// TIA Portal V19 export
FUNCTION "AI SCALING" : Void   // FC5, LAD
{ S7_Optimized_Access := 'TRUE' }
// stored: SetENOAutomatically false
   VAR_TEMP   // added for the SCL form of the ladder/FBD networks
      _w1 : Bool;
   END_VAR
BEGIN

REGION Network 1: LEVEL TRANSMITTER-101 ANALOG
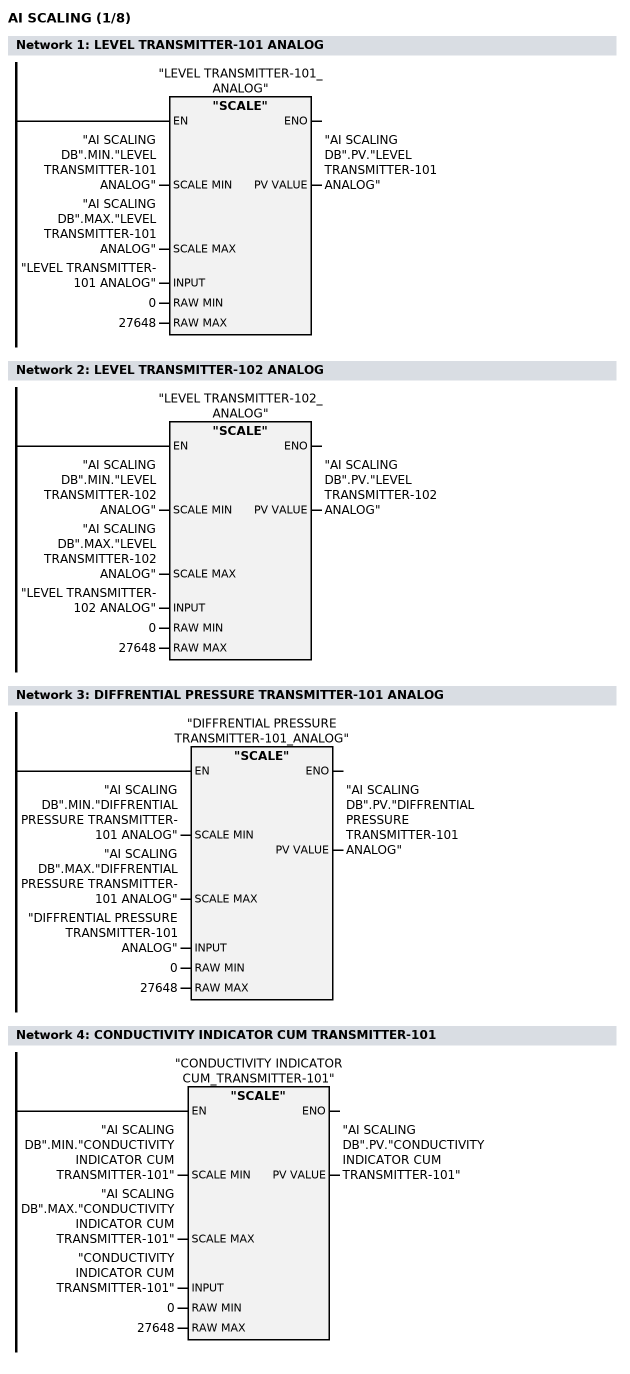
   RUNG wire#powerrail
      "LEVEL TRANSMITTER-101_ANALOG"("SCALE MIN" := "AI SCALING DB".MIN."LEVEL TRANSMITTER-101 ANALOG", "SCALE MAX" := "AI SCALING DB".MAX."LEVEL TRANSMITTER-101 ANALOG", INPUT := "LEVEL TRANSMITTER-101 ANALOG", "RAW MIN" := 0, "RAW MAX" := 27648, "PV VALUE" => "AI SCALING DB".PV."LEVEL TRANSMITTER-101 ANALOG")
   END_RUNG
   // the same network as SCL:
   "LEVEL TRANSMITTER-101_ANALOG"("SCALE MIN" := "AI SCALING DB".MIN."LEVEL TRANSMITTER-101 ANALOG",   // "SCALE"
                           "SCALE MAX" := "AI SCALING DB".MAX."LEVEL TRANSMITTER-101 ANALOG",
                           INPUT := "LEVEL TRANSMITTER-101 ANALOG",
                           "RAW MIN" := 0,
                           "RAW MAX" := 27648,
                           "PV VALUE" => "AI SCALING DB".PV."LEVEL TRANSMITTER-101 ANALOG");
END_REGION

REGION Network 2: LEVEL TRANSMITTER-102 ANALOG
   RUNG wire#powerrail
      "LEVEL TRANSMITTER-102_ANALOG"("SCALE MIN" := "AI SCALING DB".MIN."LEVEL TRANSMITTER-102 ANALOG", "SCALE MAX" := "AI SCALING DB".MAX."LEVEL TRANSMITTER-102 ANALOG", INPUT := "LEVEL TRANSMITTER-102 ANALOG", "RAW MIN" := 0, "RAW MAX" := 27648, "PV VALUE" => "AI SCALING DB".PV."LEVEL TRANSMITTER-102 ANALOG")
   END_RUNG
   // the same network as SCL:
   "LEVEL TRANSMITTER-102_ANALOG"("SCALE MIN" := "AI SCALING DB".MIN."LEVEL TRANSMITTER-102 ANALOG",   // "SCALE"
                           "SCALE MAX" := "AI SCALING DB".MAX."LEVEL TRANSMITTER-102 ANALOG",
                           INPUT := "LEVEL TRANSMITTER-102 ANALOG",
                           "RAW MIN" := 0,
                           "RAW MAX" := 27648,
                           "PV VALUE" => "AI SCALING DB".PV."LEVEL TRANSMITTER-102 ANALOG");
END_REGION

REGION Network 3: DIFFRENTIAL PRESSURE TRANSMITTER-101 ANALOG
   RUNG wire#powerrail
      "DIFFRENTIAL PRESSURE TRANSMITTER-101_ANALOG"("SCALE MIN" := "AI SCALING DB".MIN."DIFFRENTIAL PRESSURE TRANSMITTER-101 ANALOG", "SCALE MAX" := "AI SCALING DB".MAX."DIFFRENTIAL PRESSURE TRANSMITTER-101 ANALOG", INPUT := "DIFFRENTIAL PRESSURE TRANSMITTER-101 ANALOG", "RAW MIN" := 0, "RAW MAX" := 27648, "PV VALUE" => "AI SCALING DB".PV."DIFFRENTIAL PRESSURE TRANSMITTER-101 ANALOG")
   END_RUNG
   // the same network as SCL:
   "DIFFRENTIAL PRESSURE TRANSMITTER-101_ANALOG"("SCALE MIN" := "AI SCALING DB".MIN."DIFFRENTIAL PRESSURE TRANSMITTER-101 ANALOG",   // "SCALE"
                           "SCALE MAX" := "AI SCALING DB".MAX."DIFFRENTIAL PRESSURE TRANSMITTER-101 ANALOG",
                           INPUT := "DIFFRENTIAL PRESSURE TRANSMITTER-101 ANALOG",
                           "RAW MIN" := 0,
                           "RAW MAX" := 27648,
                           "PV VALUE" => "AI SCALING DB".PV."DIFFRENTIAL PRESSURE TRANSMITTER-101 ANALOG");
END_REGION

REGION Network 4: CONDUCTIVITY INDICATOR CUM TRANSMITTER-101
   RUNG wire#powerrail
      "CONDUCTIVITY INDICATOR CUM_TRANSMITTER-101"("SCALE MIN" := "AI SCALING DB".MIN."CONDUCTIVITY INDICATOR CUM TRANSMITTER-101", "SCALE MAX" := "AI SCALING DB".MAX."CONDUCTIVITY INDICATOR CUM TRANSMITTER-101", INPUT := "CONDUCTIVITY INDICATOR CUM TRANSMITTER-101", "RAW MIN" := 0, "RAW MAX" := 27648, "PV VALUE" => "AI SCALING DB".PV."CONDUCTIVITY INDICATOR CUM TRANSMITTER-101")
   END_RUNG
   // the same network as SCL:
   "CONDUCTIVITY INDICATOR CUM_TRANSMITTER-101"("SCALE MIN" := "AI SCALING DB".MIN."CONDUCTIVITY INDICATOR CUM TRANSMITTER-101",   // "SCALE"
                           "SCALE MAX" := "AI SCALING DB".MAX."CONDUCTIVITY INDICATOR CUM TRANSMITTER-101",
                           INPUT := "CONDUCTIVITY INDICATOR CUM TRANSMITTER-101",
                           "RAW MIN" := 0,
                           "RAW MAX" := 27648,
                           "PV VALUE" => "AI SCALING DB".PV."CONDUCTIVITY INDICATOR CUM TRANSMITTER-101");
END_REGION

REGION Network 5: DIFFRENTIAL PRESSURE TRANSMITTER-201
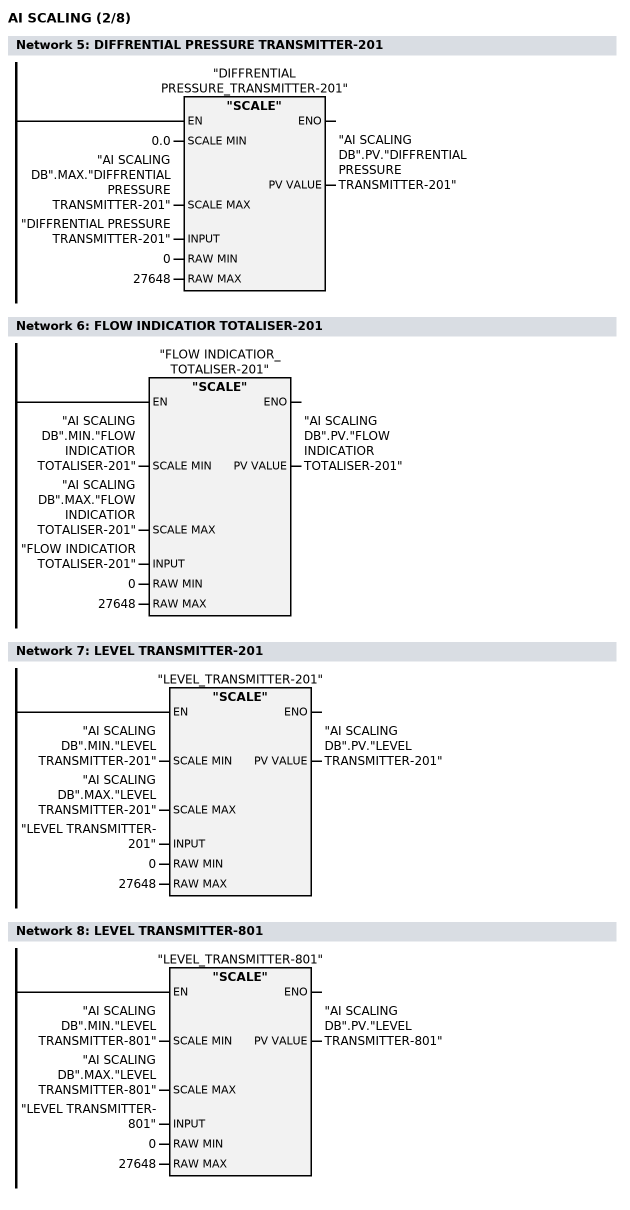
   RUNG wire#powerrail
      "DIFFRENTIAL PRESSURE_TRANSMITTER-201"("SCALE MIN" := 0.0, "SCALE MAX" := "AI SCALING DB".MAX."DIFFRENTIAL PRESSURE TRANSMITTER-201", INPUT := "DIFFRENTIAL PRESSURE TRANSMITTER-201", "RAW MIN" := 0, "RAW MAX" := 27648, "PV VALUE" => "AI SCALING DB".PV."DIFFRENTIAL PRESSURE TRANSMITTER-201")
   END_RUNG
   // the same network as SCL:
   "DIFFRENTIAL PRESSURE_TRANSMITTER-201"("SCALE MIN" := 0.0,   // "SCALE"
                           "SCALE MAX" := "AI SCALING DB".MAX."DIFFRENTIAL PRESSURE TRANSMITTER-201",
                           INPUT := "DIFFRENTIAL PRESSURE TRANSMITTER-201",
                           "RAW MIN" := 0,
                           "RAW MAX" := 27648,
                           "PV VALUE" => "AI SCALING DB".PV."DIFFRENTIAL PRESSURE TRANSMITTER-201");
END_REGION

REGION Network 6: FLOW INDICATIOR TOTALISER-201
   RUNG wire#powerrail
      "FLOW INDICATIOR_TOTALISER-201"("SCALE MIN" := "AI SCALING DB".MIN."FLOW INDICATIOR TOTALISER-201", "SCALE MAX" := "AI SCALING DB".MAX."FLOW INDICATIOR TOTALISER-201", INPUT := "FLOW INDICATIOR TOTALISER-201", "RAW MIN" := 0, "RAW MAX" := 27648, "PV VALUE" => "AI SCALING DB".PV."FLOW INDICATIOR TOTALISER-201")
   END_RUNG
   // the same network as SCL:
   "FLOW INDICATIOR_TOTALISER-201"("SCALE MIN" := "AI SCALING DB".MIN."FLOW INDICATIOR TOTALISER-201",   // "SCALE"
                           "SCALE MAX" := "AI SCALING DB".MAX."FLOW INDICATIOR TOTALISER-201",
                           INPUT := "FLOW INDICATIOR TOTALISER-201",
                           "RAW MIN" := 0,
                           "RAW MAX" := 27648,
                           "PV VALUE" => "AI SCALING DB".PV."FLOW INDICATIOR TOTALISER-201");
END_REGION

REGION Network 7: LEVEL TRANSMITTER-201
   RUNG wire#powerrail
      "LEVEL_TRANSMITTER-201"("SCALE MIN" := "AI SCALING DB".MIN."LEVEL TRANSMITTER-201", "SCALE MAX" := "AI SCALING DB".MAX."LEVEL TRANSMITTER-201", INPUT := "LEVEL TRANSMITTER-201", "RAW MIN" := 0, "RAW MAX" := 27648, "PV VALUE" => "AI SCALING DB".PV."LEVEL TRANSMITTER-201")
   END_RUNG
   // the same network as SCL:
   "LEVEL_TRANSMITTER-201"("SCALE MIN" := "AI SCALING DB".MIN."LEVEL TRANSMITTER-201",   // "SCALE"
                           "SCALE MAX" := "AI SCALING DB".MAX."LEVEL TRANSMITTER-201",
                           INPUT := "LEVEL TRANSMITTER-201",
                           "RAW MIN" := 0,
                           "RAW MAX" := 27648,
                           "PV VALUE" => "AI SCALING DB".PV."LEVEL TRANSMITTER-201");
END_REGION

REGION Network 8: LEVEL TRANSMITTER-801
   RUNG wire#powerrail
      "LEVEL_TRANSMITTER-801"("SCALE MIN" := "AI SCALING DB".MIN."LEVEL TRANSMITTER-801", "SCALE MAX" := "AI SCALING DB".MAX."LEVEL TRANSMITTER-801", INPUT := "LEVEL TRANSMITTER-801", "RAW MIN" := 0, "RAW MAX" := 27648, "PV VALUE" => "AI SCALING DB".PV."LEVEL TRANSMITTER-801")
   END_RUNG
   // the same network as SCL:
   "LEVEL_TRANSMITTER-801"("SCALE MIN" := "AI SCALING DB".MIN."LEVEL TRANSMITTER-801",   // "SCALE"
                           "SCALE MAX" := "AI SCALING DB".MAX."LEVEL TRANSMITTER-801",
                           INPUT := "LEVEL TRANSMITTER-801",
                           "RAW MIN" := 0,
                           "RAW MAX" := 27648,
                           "PV VALUE" => "AI SCALING DB".PV."LEVEL TRANSMITTER-801");
END_REGION

REGION Network 9: RESISTIVITY CUM TRANSMITTER 601
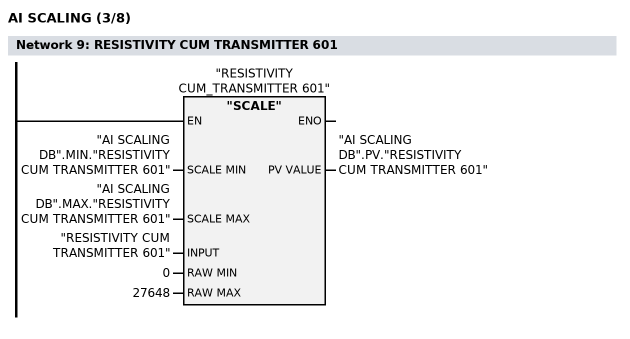
   RUNG wire#powerrail
      "RESISTIVITY CUM_TRANSMITTER 601"("SCALE MIN" := "AI SCALING DB".MIN."RESISTIVITY CUM TRANSMITTER 601", "SCALE MAX" := "AI SCALING DB".MAX."RESISTIVITY CUM TRANSMITTER 601", INPUT := "RESISTIVITY CUM TRANSMITTER 601", "RAW MIN" := 0, "RAW MAX" := 27648, "PV VALUE" => "AI SCALING DB".PV."RESISTIVITY CUM TRANSMITTER 601")
   END_RUNG
   // the same network as SCL:
   "RESISTIVITY CUM_TRANSMITTER 601"("SCALE MIN" := "AI SCALING DB".MIN."RESISTIVITY CUM TRANSMITTER 601",   // "SCALE"
                           "SCALE MAX" := "AI SCALING DB".MAX."RESISTIVITY CUM TRANSMITTER 601",
                           INPUT := "RESISTIVITY CUM TRANSMITTER 601",
                           "RAW MIN" := 0,
                           "RAW MAX" := 27648,
                           "PV VALUE" => "AI SCALING DB".PV."RESISTIVITY CUM TRANSMITTER 601");
END_REGION

REGION Network 10: PRESSURE TRANSMITTER 601
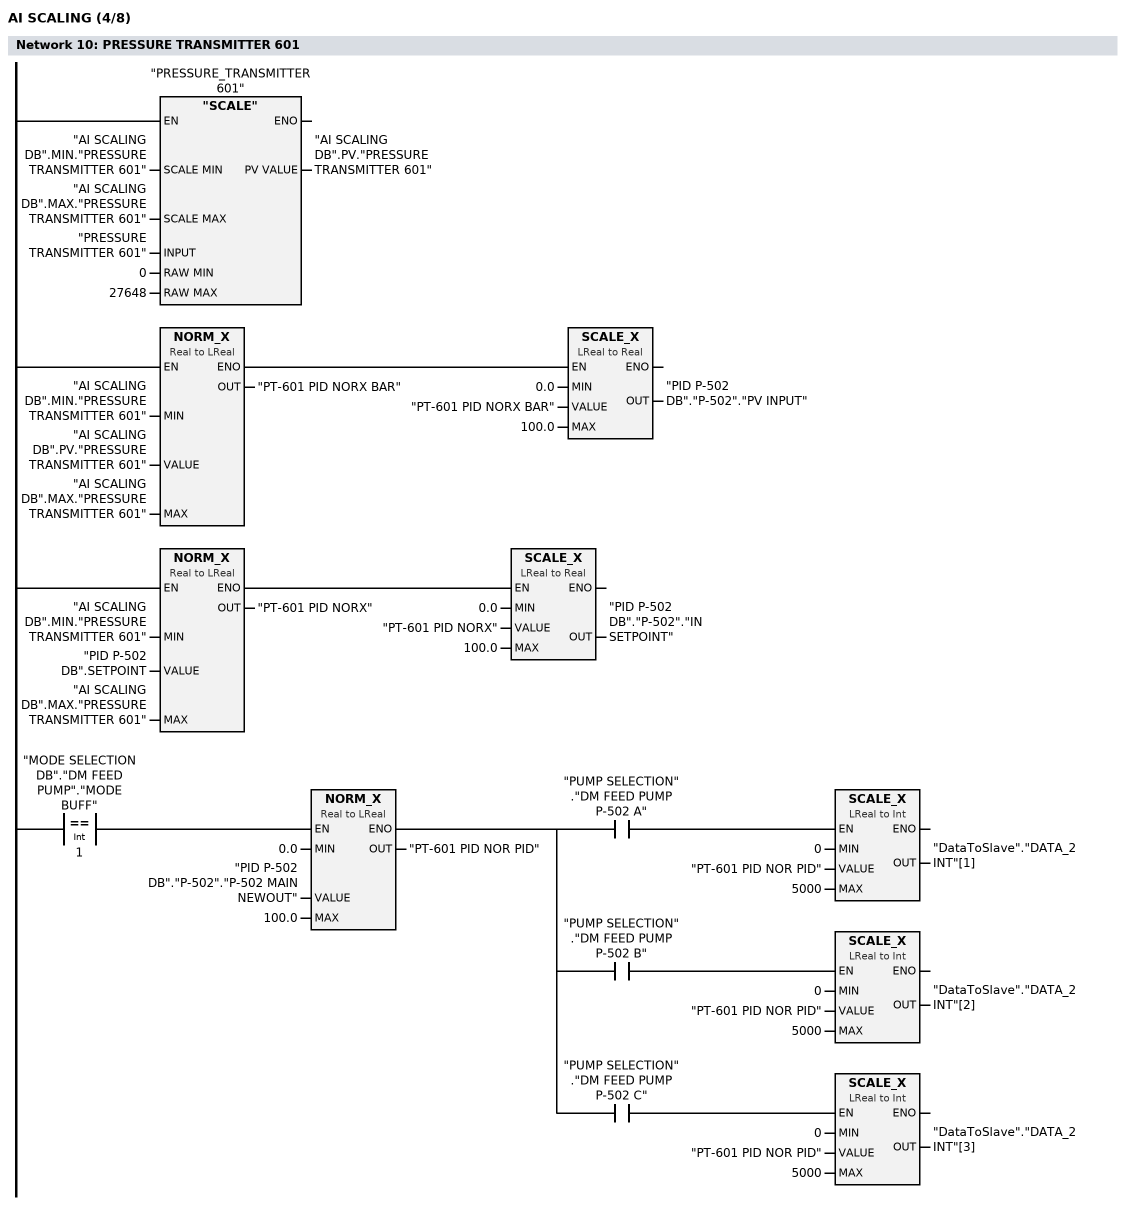
   RUNG wire#powerrail
      "PRESSURE_TRANSMITTER 601"("SCALE MIN" := "AI SCALING DB".MIN."PRESSURE TRANSMITTER 601", "SCALE MAX" := "AI SCALING DB".MAX."PRESSURE TRANSMITTER 601", INPUT := "PRESSURE TRANSMITTER 601", "RAW MIN" := 0, "RAW MAX" := 27648, "PV VALUE" => "AI SCALING DB".PV."PRESSURE TRANSMITTER 601")
   END_RUNG
   RUNG wire#powerrail
      { S7_Templates := "[SrcType := Real, DestType := LReal]" } Normalize(min := "AI SCALING DB".MIN."PRESSURE TRANSMITTER 601", value := "AI SCALING DB".PV."PRESSURE TRANSMITTER 601", max := "AI SCALING DB".MAX."PRESSURE TRANSMITTER 601", out => "PT-601 PID NORX BAR")
      { S7_Templates := "[SrcType := LReal, DestType := Real]" } Scale(min := 0.0, value := "PT-601 PID NORX BAR", max := 100.0, out => "PID P-502 DB"."P-502"."PV INPUT")
   END_RUNG
   RUNG wire#powerrail
      { S7_Templates := "[SrcType := Real, DestType := LReal]" } Normalize(min := "AI SCALING DB".MIN."PRESSURE TRANSMITTER 601", value := "PID P-502 DB".SETPOINT, max := "AI SCALING DB".MAX."PRESSURE TRANSMITTER 601", out => "PT-601 PID NORX")
      { S7_Templates := "[SrcType := LReal, DestType := Real]" } Scale(min := 0.0, value := "PT-601 PID NORX", max := 100.0, out => "PID P-502 DB"."P-502"."IN SETPOINT")
   END_RUNG
   RUNG wire#powerrail
      { S7_Templates := "SrcType := Int" } EQ_Contact(in1 := "MODE SELECTION DB"."DM FEED PUMP"."MODE BUFF", in2 := 1)
      { S7_Templates := "[SrcType := Real, DestType := LReal]" } Normalize(min := 0.0, value := "PID P-502 DB"."P-502"."P-502 MAIN NEWOUT", max := 100.0, out => "PT-601 PID NOR PID")
      wire#w1
      Contact( "PUMP SELECTION"."DM FEED PUMP P-502 A" )
      { S7_Templates := "[SrcType := LReal, DestType := Int]" } Scale(min := 0, value := "PT-601 PID NOR PID", max := 5000, out => "DataToSlave"."DATA_2 INT"[1])
   END_RUNG
   RUNG wire#w1
      Contact( "PUMP SELECTION"."DM FEED PUMP P-502 B" )
      { S7_Templates := "[SrcType := LReal, DestType := Int]" } Scale(min := 0, value := "PT-601 PID NOR PID", max := 5000, out => "DataToSlave"."DATA_2 INT"[2])
   END_RUNG
   RUNG wire#w1
      Contact( "PUMP SELECTION"."DM FEED PUMP P-502 C" )
      { S7_Templates := "[SrcType := LReal, DestType := Int]" } Scale(min := 0, value := "PT-601 PID NOR PID", max := 5000, out => "DataToSlave"."DATA_2 INT"[3])
   END_RUNG
   // the same network as SCL:
   "PRESSURE_TRANSMITTER 601"("SCALE MIN" := "AI SCALING DB".MIN."PRESSURE TRANSMITTER 601",   // "SCALE"
                           "SCALE MAX" := "AI SCALING DB".MAX."PRESSURE TRANSMITTER 601",
                           INPUT := "PRESSURE TRANSMITTER 601",
                           "RAW MIN" := 0,
                           "RAW MAX" := 27648,
                           "PV VALUE" => "AI SCALING DB".PV."PRESSURE TRANSMITTER 601");
   "PT-601 PID NORX BAR" := NORM_X(MIN := "AI SCALING DB".MIN."PRESSURE TRANSMITTER 601", VALUE := "AI SCALING DB".PV."PRESSURE TRANSMITTER 601", MAX := "AI SCALING DB".MAX."PRESSURE TRANSMITTER 601");
   "PID P-502 DB"."P-502"."PV INPUT" := SCALE_X(MIN := 0.0, VALUE := "PT-601 PID NORX BAR", MAX := 100.0);
   "PT-601 PID NORX" := NORM_X(MIN := "AI SCALING DB".MIN."PRESSURE TRANSMITTER 601", VALUE := "PID P-502 DB".SETPOINT, MAX := "AI SCALING DB".MAX."PRESSURE TRANSMITTER 601");
   "PID P-502 DB"."P-502"."IN SETPOINT" := SCALE_X(MIN := 0.0, VALUE := "PT-601 PID NORX", MAX := 100.0);
   #_w1 := "MODE SELECTION DB"."DM FEED PUMP"."MODE BUFF" = 1;
   IF #_w1 THEN
       "PT-601 PID NOR PID" := NORM_X(MIN := 0.0, VALUE := "PID P-502 DB"."P-502"."P-502 MAIN NEWOUT", MAX := 100.0);
   END_IF;
   IF #_w1 AND "PUMP SELECTION"."DM FEED PUMP P-502 A" THEN
       "DataToSlave"."DATA_2 INT"[1] := SCALE_X(MIN := 0, VALUE := "PT-601 PID NOR PID", MAX := 5000);
   END_IF;
   IF #_w1 AND "PUMP SELECTION"."DM FEED PUMP P-502 B" THEN
       "DataToSlave"."DATA_2 INT"[2] := SCALE_X(MIN := 0, VALUE := "PT-601 PID NOR PID", MAX := 5000);
   END_IF;
   IF #_w1 AND "PUMP SELECTION"."DM FEED PUMP P-502 C" THEN
       "DataToSlave"."DATA_2 INT"[3] := SCALE_X(MIN := 0, VALUE := "PT-601 PID NOR PID", MAX := 5000);
   END_IF;
END_REGION

REGION Network 11: FLOW INDICATIOR TOTALISER 601
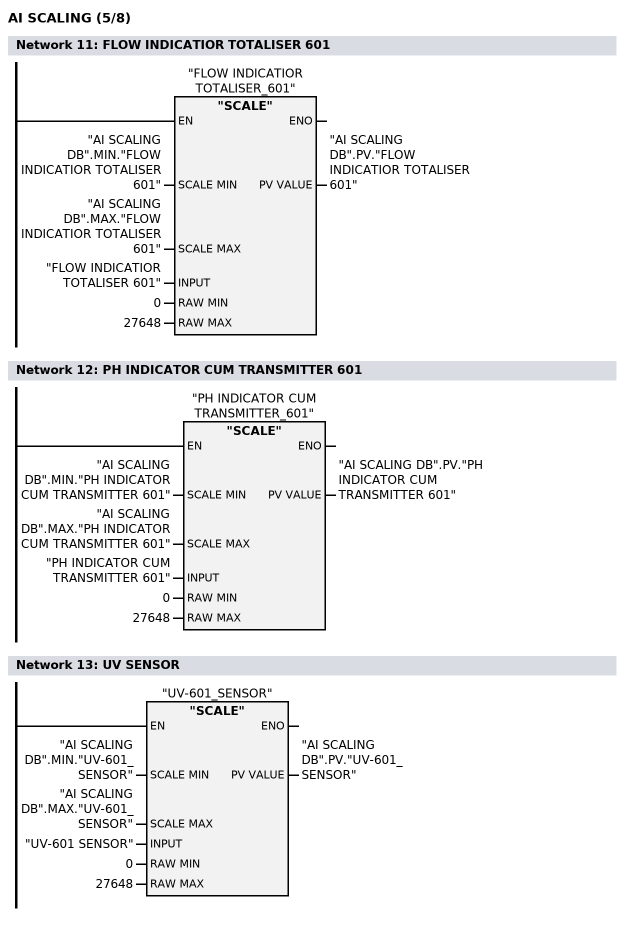
   RUNG wire#powerrail
      "FLOW INDICATIOR TOTALISER_601"("SCALE MIN" := "AI SCALING DB".MIN."FLOW INDICATIOR TOTALISER 601", "SCALE MAX" := "AI SCALING DB".MAX."FLOW INDICATIOR TOTALISER 601", INPUT := "FLOW INDICATIOR TOTALISER 601", "RAW MIN" := 0, "RAW MAX" := 27648, "PV VALUE" => "AI SCALING DB".PV."FLOW INDICATIOR TOTALISER 601")
   END_RUNG
   // the same network as SCL:
   "FLOW INDICATIOR TOTALISER_601"("SCALE MIN" := "AI SCALING DB".MIN."FLOW INDICATIOR TOTALISER 601",   // "SCALE"
                           "SCALE MAX" := "AI SCALING DB".MAX."FLOW INDICATIOR TOTALISER 601",
                           INPUT := "FLOW INDICATIOR TOTALISER 601",
                           "RAW MIN" := 0,
                           "RAW MAX" := 27648,
                           "PV VALUE" => "AI SCALING DB".PV."FLOW INDICATIOR TOTALISER 601");
END_REGION

REGION Network 12: PH INDICATOR CUM TRANSMITTER 601
   RUNG wire#powerrail
      "PH INDICATOR CUM TRANSMITTER_601"("SCALE MIN" := "AI SCALING DB".MIN."PH INDICATOR CUM TRANSMITTER 601", "SCALE MAX" := "AI SCALING DB".MAX."PH INDICATOR CUM TRANSMITTER 601", INPUT := "PH INDICATOR CUM TRANSMITTER 601", "RAW MIN" := 0, "RAW MAX" := 27648, "PV VALUE" => "AI SCALING DB".PV."PH INDICATOR CUM TRANSMITTER 601")
   END_RUNG
   // the same network as SCL:
   "PH INDICATOR CUM TRANSMITTER_601"("SCALE MIN" := "AI SCALING DB".MIN."PH INDICATOR CUM TRANSMITTER 601",   // "SCALE"
                           "SCALE MAX" := "AI SCALING DB".MAX."PH INDICATOR CUM TRANSMITTER 601",
                           INPUT := "PH INDICATOR CUM TRANSMITTER 601",
                           "RAW MIN" := 0,
                           "RAW MAX" := 27648,
                           "PV VALUE" => "AI SCALING DB".PV."PH INDICATOR CUM TRANSMITTER 601");
END_REGION

REGION Network 13: UV SENSOR
   RUNG wire#powerrail
      "UV-601_SENSOR"("SCALE MIN" := "AI SCALING DB".MIN."UV-601_SENSOR", "SCALE MAX" := "AI SCALING DB".MAX."UV-601_SENSOR", INPUT := "UV-601 SENSOR", "RAW MIN" := 0, "RAW MAX" := 27648, "PV VALUE" => "AI SCALING DB".PV."UV-601_SENSOR")
   END_RUNG
   // the same network as SCL:
   "UV-601_SENSOR"("SCALE MIN" := "AI SCALING DB".MIN."UV-601_SENSOR",   // "SCALE"
                   "SCALE MAX" := "AI SCALING DB".MAX."UV-601_SENSOR",
                   INPUT := "UV-601 SENSOR",
                   "RAW MIN" := 0,
                   "RAW MAX" := 27648,
                   "PV VALUE" => "AI SCALING DB".PV."UV-601_SENSOR");
END_REGION

REGION Network 16: LT-101 BUFFER
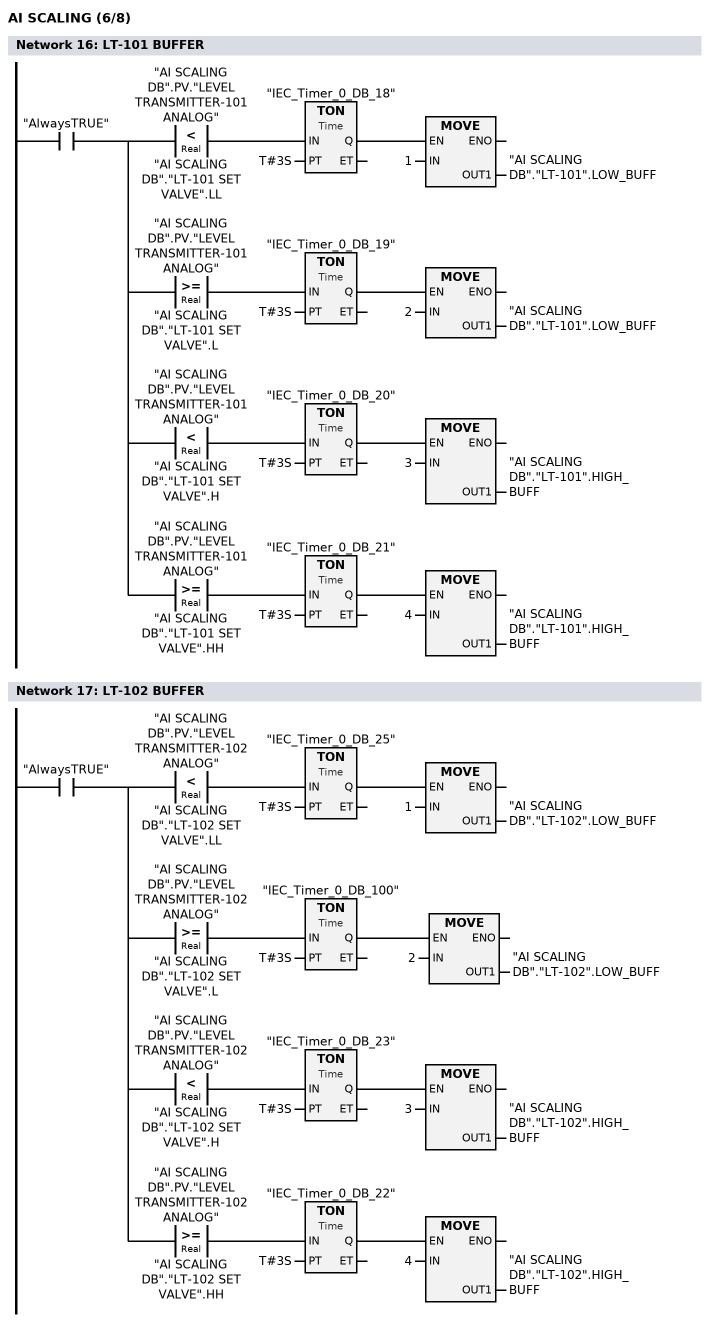
   RUNG wire#powerrail
      Contact( "AlwaysTRUE" )
      wire#w1
      { S7_Templates := "SrcType := Real" } LT_Contact(in1 := "AI SCALING DB".PV."LEVEL TRANSMITTER-101 ANALOG", in2 := "AI SCALING DB"."LT-101 SET VALVE".LL)
      { S7_Templates := "time_type := Time" } "IEC_Timer_0_DB_18".TON(pt := T#3S, et =>)
      Move(in := 1, out1 => "AI SCALING DB"."LT-101".LOW_BUFF)
   END_RUNG
   RUNG wire#w1
      { S7_Templates := "SrcType := Real" } GE_Contact(in1 := "AI SCALING DB".PV."LEVEL TRANSMITTER-101 ANALOG", in2 := "AI SCALING DB"."LT-101 SET VALVE".L)
      { S7_Templates := "time_type := Time" } "IEC_Timer_0_DB_19".TON(pt := T#3S, et =>)
      Move(in := 2, out1 => "AI SCALING DB"."LT-101".LOW_BUFF)
   END_RUNG
   RUNG wire#w1
      { S7_Templates := "SrcType := Real" } LT_Contact(in1 := "AI SCALING DB".PV."LEVEL TRANSMITTER-101 ANALOG", in2 := "AI SCALING DB"."LT-101 SET VALVE".H)
      { S7_Templates := "time_type := Time" } "IEC_Timer_0_DB_20".TON(pt := T#3S, et =>)
      Move(in := 3, out1 => "AI SCALING DB"."LT-101".HIGH_BUFF)
   END_RUNG
   RUNG wire#w1
      { S7_Templates := "SrcType := Real" } GE_Contact(in1 := "AI SCALING DB".PV."LEVEL TRANSMITTER-101 ANALOG", in2 := "AI SCALING DB"."LT-101 SET VALVE".HH)
      { S7_Templates := "time_type := Time" } "IEC_Timer_0_DB_21".TON(pt := T#3S, et =>)
      Move(in := 4, out1 => "AI SCALING DB"."LT-101".HIGH_BUFF)
   END_RUNG
   // the same network as SCL:
   "IEC_Timer_0_DB_18".TON(IN := "AlwaysTRUE" AND ("AI SCALING DB".PV."LEVEL TRANSMITTER-101 ANALOG" < "AI SCALING DB"."LT-101 SET VALVE".LL),
                           PT := T#3S);
   IF "IEC_Timer_0_DB_18".Q THEN "AI SCALING DB"."LT-101".LOW_BUFF := 1; END_IF;
   "IEC_Timer_0_DB_19".TON(IN := "AlwaysTRUE" AND ("AI SCALING DB".PV."LEVEL TRANSMITTER-101 ANALOG" >= "AI SCALING DB"."LT-101 SET VALVE".L),
                           PT := T#3S);
   IF "IEC_Timer_0_DB_19".Q THEN "AI SCALING DB"."LT-101".LOW_BUFF := 2; END_IF;
   "IEC_Timer_0_DB_20".TON(IN := "AlwaysTRUE" AND ("AI SCALING DB".PV."LEVEL TRANSMITTER-101 ANALOG" < "AI SCALING DB"."LT-101 SET VALVE".H),
                           PT := T#3S);
   IF "IEC_Timer_0_DB_20".Q THEN "AI SCALING DB"."LT-101".HIGH_BUFF := 3; END_IF;
   "IEC_Timer_0_DB_21".TON(IN := "AlwaysTRUE" AND ("AI SCALING DB".PV."LEVEL TRANSMITTER-101 ANALOG" >= "AI SCALING DB"."LT-101 SET VALVE".HH),
                           PT := T#3S);
   IF "IEC_Timer_0_DB_21".Q THEN "AI SCALING DB"."LT-101".HIGH_BUFF := 4; END_IF;
END_REGION

REGION Network 17: LT-102 BUFFER
   RUNG wire#powerrail
      Contact( "AlwaysTRUE" )
      wire#w1
      { S7_Templates := "SrcType := Real" } LT_Contact(in1 := "AI SCALING DB".PV."LEVEL TRANSMITTER-102 ANALOG", in2 := "AI SCALING DB"."LT-102 SET VALVE".LL)
      { S7_Templates := "time_type := Time" } "IEC_Timer_0_DB_25".TON(pt := T#3S, et =>)
      Move(in := 1, out1 => "AI SCALING DB"."LT-102".LOW_BUFF)
   END_RUNG
   RUNG wire#w1
      { S7_Templates := "SrcType := Real" } GE_Contact(in1 := "AI SCALING DB".PV."LEVEL TRANSMITTER-102 ANALOG", in2 := "AI SCALING DB"."LT-102 SET VALVE".L)
      { S7_Templates := "time_type := Time" } "IEC_Timer_0_DB_100".TON(pt := T#3S, et =>)
      Move(in := 2, out1 => "AI SCALING DB"."LT-102".LOW_BUFF)
   END_RUNG
   RUNG wire#w1
      { S7_Templates := "SrcType := Real" } LT_Contact(in1 := "AI SCALING DB".PV."LEVEL TRANSMITTER-102 ANALOG", in2 := "AI SCALING DB"."LT-102 SET VALVE".H)
      { S7_Templates := "time_type := Time" } "IEC_Timer_0_DB_23".TON(pt := T#3S, et =>)
      Move(in := 3, out1 => "AI SCALING DB"."LT-102".HIGH_BUFF)
   END_RUNG
   RUNG wire#w1
      { S7_Templates := "SrcType := Real" } GE_Contact(in1 := "AI SCALING DB".PV."LEVEL TRANSMITTER-102 ANALOG", in2 := "AI SCALING DB"."LT-102 SET VALVE".HH)
      { S7_Templates := "time_type := Time" } "IEC_Timer_0_DB_22".TON(pt := T#3S, et =>)
      Move(in := 4, out1 => "AI SCALING DB"."LT-102".HIGH_BUFF)
   END_RUNG
   // the same network as SCL:
   "IEC_Timer_0_DB_25".TON(IN := "AlwaysTRUE" AND ("AI SCALING DB".PV."LEVEL TRANSMITTER-102 ANALOG" < "AI SCALING DB"."LT-102 SET VALVE".LL),
                           PT := T#3S);
   IF "IEC_Timer_0_DB_25".Q THEN "AI SCALING DB"."LT-102".LOW_BUFF := 1; END_IF;
   "IEC_Timer_0_DB_100".TON(IN := "AlwaysTRUE" AND ("AI SCALING DB".PV."LEVEL TRANSMITTER-102 ANALOG" >= "AI SCALING DB"."LT-102 SET VALVE".L),
                           PT := T#3S);
   IF "IEC_Timer_0_DB_100".Q THEN "AI SCALING DB"."LT-102".LOW_BUFF := 2; END_IF;
   "IEC_Timer_0_DB_23".TON(IN := "AlwaysTRUE" AND ("AI SCALING DB".PV."LEVEL TRANSMITTER-102 ANALOG" < "AI SCALING DB"."LT-102 SET VALVE".H),
                           PT := T#3S);
   IF "IEC_Timer_0_DB_23".Q THEN "AI SCALING DB"."LT-102".HIGH_BUFF := 3; END_IF;
   "IEC_Timer_0_DB_22".TON(IN := "AlwaysTRUE" AND ("AI SCALING DB".PV."LEVEL TRANSMITTER-102 ANALOG" >= "AI SCALING DB"."LT-102 SET VALVE".HH),
                           PT := T#3S);
   IF "IEC_Timer_0_DB_22".Q THEN "AI SCALING DB"."LT-102".HIGH_BUFF := 4; END_IF;
END_REGION

REGION Network 18: LT-201 BUFFER
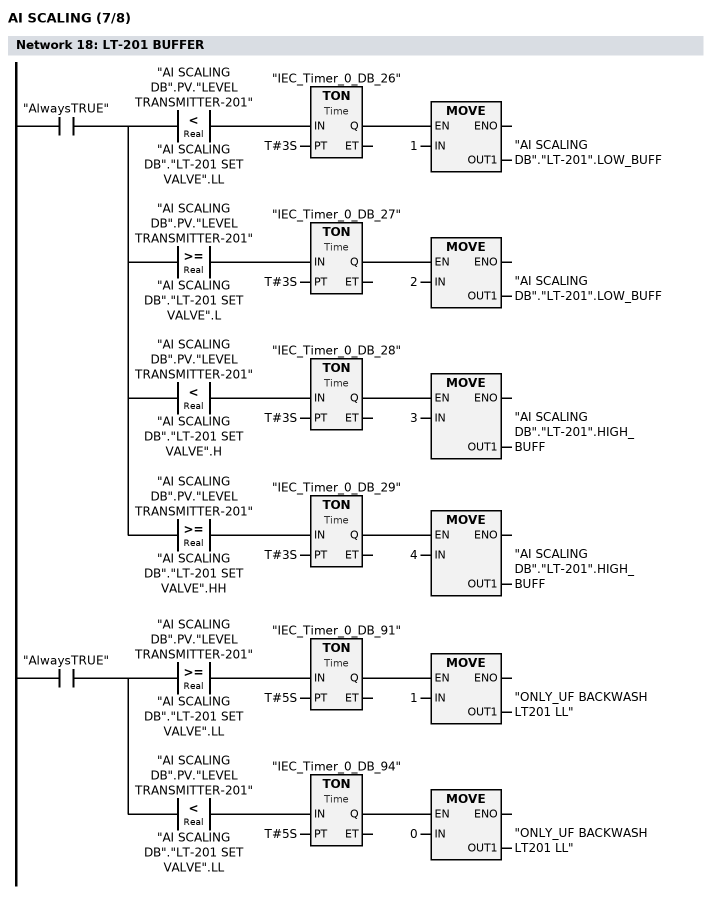
   RUNG wire#powerrail
      Contact( "AlwaysTRUE" )
      wire#w1
      { S7_Templates := "SrcType := Real" } LT_Contact(in1 := "AI SCALING DB".PV."LEVEL TRANSMITTER-201", in2 := "AI SCALING DB"."LT-201 SET VALVE".LL)
      { S7_Templates := "time_type := Time" } "IEC_Timer_0_DB_26".TON(pt := T#3S, et =>)
      Move(in := 1, out1 => "AI SCALING DB"."LT-201".LOW_BUFF)
   END_RUNG
   RUNG wire#w1
      { S7_Templates := "SrcType := Real" } GE_Contact(in1 := "AI SCALING DB".PV."LEVEL TRANSMITTER-201", in2 := "AI SCALING DB"."LT-201 SET VALVE".L)
      { S7_Templates := "time_type := Time" } "IEC_Timer_0_DB_27".TON(pt := T#3S, et =>)
      Move(in := 2, out1 => "AI SCALING DB"."LT-201".LOW_BUFF)
   END_RUNG
   RUNG wire#w1
      { S7_Templates := "SrcType := Real" } LT_Contact(in1 := "AI SCALING DB".PV."LEVEL TRANSMITTER-201", in2 := "AI SCALING DB"."LT-201 SET VALVE".H)
      { S7_Templates := "time_type := Time" } "IEC_Timer_0_DB_28".TON(pt := T#3S, et =>)
      Move(in := 3, out1 => "AI SCALING DB"."LT-201".HIGH_BUFF)
   END_RUNG
   RUNG wire#w1
      { S7_Templates := "SrcType := Real" } GE_Contact(in1 := "AI SCALING DB".PV."LEVEL TRANSMITTER-201", in2 := "AI SCALING DB"."LT-201 SET VALVE".HH)
      { S7_Templates := "time_type := Time" } "IEC_Timer_0_DB_29".TON(pt := T#3S, et =>)
      Move(in := 4, out1 => "AI SCALING DB"."LT-201".HIGH_BUFF)
   END_RUNG
   RUNG wire#powerrail
      Contact( "AlwaysTRUE" )
      wire#w2
      { S7_Templates := "SrcType := Real" } GE_Contact(in1 := "AI SCALING DB".PV."LEVEL TRANSMITTER-201", in2 := "AI SCALING DB"."LT-201 SET VALVE".LL)
      { S7_Templates := "time_type := Time" } "IEC_Timer_0_DB_91".TON(pt := T#5S, et =>)
      Move(in := 1, out1 => "ONLY_UF BACKWASH LT201 LL")
   END_RUNG
   RUNG wire#w2
      { S7_Templates := "SrcType := Real" } LT_Contact(in1 := "AI SCALING DB".PV."LEVEL TRANSMITTER-201", in2 := "AI SCALING DB"."LT-201 SET VALVE".LL)
      { S7_Templates := "time_type := Time" } "IEC_Timer_0_DB_94".TON(pt := T#5S, et =>)
      Move(in := 0, out1 => "ONLY_UF BACKWASH LT201 LL")
   END_RUNG
   // the same network as SCL:
   "IEC_Timer_0_DB_26".TON(IN := "AlwaysTRUE" AND ("AI SCALING DB".PV."LEVEL TRANSMITTER-201" < "AI SCALING DB"."LT-201 SET VALVE".LL),
                           PT := T#3S);
   IF "IEC_Timer_0_DB_26".Q THEN "AI SCALING DB"."LT-201".LOW_BUFF := 1; END_IF;
   "IEC_Timer_0_DB_27".TON(IN := "AlwaysTRUE" AND ("AI SCALING DB".PV."LEVEL TRANSMITTER-201" >= "AI SCALING DB"."LT-201 SET VALVE".L),
                           PT := T#3S);
   IF "IEC_Timer_0_DB_27".Q THEN "AI SCALING DB"."LT-201".LOW_BUFF := 2; END_IF;
   "IEC_Timer_0_DB_28".TON(IN := "AlwaysTRUE" AND ("AI SCALING DB".PV."LEVEL TRANSMITTER-201" < "AI SCALING DB"."LT-201 SET VALVE".H),
                           PT := T#3S);
   IF "IEC_Timer_0_DB_28".Q THEN "AI SCALING DB"."LT-201".HIGH_BUFF := 3; END_IF;
   "IEC_Timer_0_DB_29".TON(IN := "AlwaysTRUE" AND ("AI SCALING DB".PV."LEVEL TRANSMITTER-201" >= "AI SCALING DB"."LT-201 SET VALVE".HH),
                           PT := T#3S);
   IF "IEC_Timer_0_DB_29".Q THEN "AI SCALING DB"."LT-201".HIGH_BUFF := 4; END_IF;
   "IEC_Timer_0_DB_91".TON(IN := "AlwaysTRUE" AND ("AI SCALING DB".PV."LEVEL TRANSMITTER-201" >= "AI SCALING DB"."LT-201 SET VALVE".LL),
                           PT := T#5S);
   IF "IEC_Timer_0_DB_91".Q THEN "ONLY_UF BACKWASH LT201 LL" := 1; END_IF;
   "IEC_Timer_0_DB_94".TON(IN := "AlwaysTRUE" AND ("AI SCALING DB".PV."LEVEL TRANSMITTER-201" < "AI SCALING DB"."LT-201 SET VALVE".LL),
                           PT := T#5S);
   IF "IEC_Timer_0_DB_94".Q THEN "ONLY_UF BACKWASH LT201 LL" := 0; END_IF;
END_REGION

REGION Network 19: LT-801 BUFFER
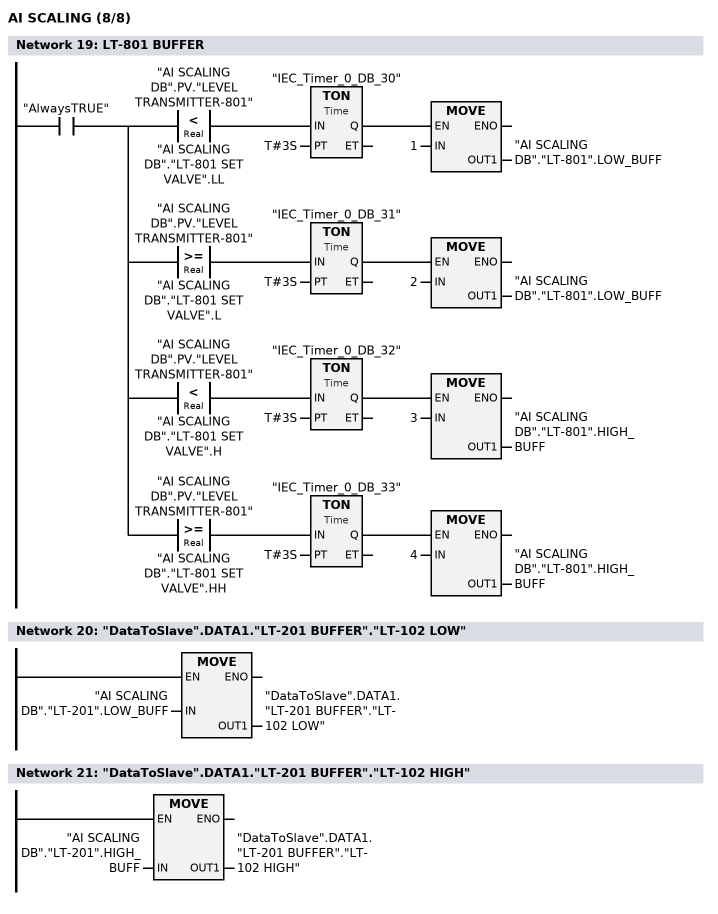
   RUNG wire#powerrail
      Contact( "AlwaysTRUE" )
      wire#w1
      { S7_Templates := "SrcType := Real" } LT_Contact(in1 := "AI SCALING DB".PV."LEVEL TRANSMITTER-801", in2 := "AI SCALING DB"."LT-801 SET VALVE".LL)
      { S7_Templates := "time_type := Time" } "IEC_Timer_0_DB_30".TON(pt := T#3S, et =>)
      Move(in := 1, out1 => "AI SCALING DB"."LT-801".LOW_BUFF)
   END_RUNG
   RUNG wire#w1
      { S7_Templates := "SrcType := Real" } GE_Contact(in1 := "AI SCALING DB".PV."LEVEL TRANSMITTER-801", in2 := "AI SCALING DB"."LT-801 SET VALVE".L)
      { S7_Templates := "time_type := Time" } "IEC_Timer_0_DB_31".TON(pt := T#3S, et =>)
      Move(in := 2, out1 => "AI SCALING DB"."LT-801".LOW_BUFF)
   END_RUNG
   RUNG wire#w1
      { S7_Templates := "SrcType := Real" } LT_Contact(in1 := "AI SCALING DB".PV."LEVEL TRANSMITTER-801", in2 := "AI SCALING DB"."LT-801 SET VALVE".H)
      { S7_Templates := "time_type := Time" } "IEC_Timer_0_DB_32".TON(pt := T#3S, et =>)
      Move(in := 3, out1 => "AI SCALING DB"."LT-801".HIGH_BUFF)
   END_RUNG
   RUNG wire#w1
      { S7_Templates := "SrcType := Real" } GE_Contact(in1 := "AI SCALING DB".PV."LEVEL TRANSMITTER-801", in2 := "AI SCALING DB"."LT-801 SET VALVE".HH)
      { S7_Templates := "time_type := Time" } "IEC_Timer_0_DB_33".TON(pt := T#3S, et =>)
      Move(in := 4, out1 => "AI SCALING DB"."LT-801".HIGH_BUFF)
   END_RUNG
   // the same network as SCL:
   "IEC_Timer_0_DB_30".TON(IN := "AlwaysTRUE" AND ("AI SCALING DB".PV."LEVEL TRANSMITTER-801" < "AI SCALING DB"."LT-801 SET VALVE".LL),
                           PT := T#3S);
   IF "IEC_Timer_0_DB_30".Q THEN "AI SCALING DB"."LT-801".LOW_BUFF := 1; END_IF;
   "IEC_Timer_0_DB_31".TON(IN := "AlwaysTRUE" AND ("AI SCALING DB".PV."LEVEL TRANSMITTER-801" >= "AI SCALING DB"."LT-801 SET VALVE".L),
                           PT := T#3S);
   IF "IEC_Timer_0_DB_31".Q THEN "AI SCALING DB"."LT-801".LOW_BUFF := 2; END_IF;
   "IEC_Timer_0_DB_32".TON(IN := "AlwaysTRUE" AND ("AI SCALING DB".PV."LEVEL TRANSMITTER-801" < "AI SCALING DB"."LT-801 SET VALVE".H),
                           PT := T#3S);
   IF "IEC_Timer_0_DB_32".Q THEN "AI SCALING DB"."LT-801".HIGH_BUFF := 3; END_IF;
   "IEC_Timer_0_DB_33".TON(IN := "AlwaysTRUE" AND ("AI SCALING DB".PV."LEVEL TRANSMITTER-801" >= "AI SCALING DB"."LT-801 SET VALVE".HH),
                           PT := T#3S);
   IF "IEC_Timer_0_DB_33".Q THEN "AI SCALING DB"."LT-801".HIGH_BUFF := 4; END_IF;
END_REGION

REGION Network 20: "DataToSlave".DATA1."LT-201 BUFFER"."LT-102 LOW"
   RUNG wire#powerrail
      Move(in := "AI SCALING DB"."LT-201".LOW_BUFF, out1 => "DataToSlave".DATA1."LT-201 BUFFER"."LT-102 LOW")
   END_RUNG
   // the same network as SCL:
   "DataToSlave".DATA1."LT-201 BUFFER"."LT-102 LOW" := "AI SCALING DB"."LT-201".LOW_BUFF;
END_REGION

REGION Network 21: "DataToSlave".DATA1."LT-201 BUFFER"."LT-102 HIGH"
   RUNG wire#powerrail
      Move(in := "AI SCALING DB"."LT-201".HIGH_BUFF, out1 => "DataToSlave".DATA1."LT-201 BUFFER"."LT-102 HIGH")
   END_RUNG
   // the same network as SCL:
   "DataToSlave".DATA1."LT-201 BUFFER"."LT-102 HIGH" := "AI SCALING DB"."LT-201".HIGH_BUFF;
END_REGION
END_FUNCTION
